{attribute 'qualified_only'}
{attribute 'strict'}
TYPE SegmentType :
(
	Location := 0,
  LinePoints,
  CatmulRomPoints
);
END_TYPE

(* stored: Version 1.1.0.1
   DUT SegmentType: Id {f08d08a4-ada9-438a-a438-c698fd156174} *)
